FUNCTION_BLOCK FB_Tc3EventRead IMPLEMENTS InterfaceEventViewer
VAR CONSTANT
	DISP_ROWS : UDINT := 80;
END_VAR
VAR_INPUT
	tzinfo : ST_TimeZoneInformation;
END_VAR
VAR_OUTPUT
	stAlarmEvents	: ARRAY [1..DISP_ROWS] OF ST_ReadEventW;
	stAlarmhistory 	: ARRAY [1..DISP_ROWS] OF ST_ReadEventW;
END_VAR
VAR
	row : UDINT := 1;
END_VAR

METHOD PRIVATE _create_current_table : BOOL
VAR_INPUT
	event_container : REFERENCE TO EventContainer;
	row		: UDINT;
	stDate	: STRING;
	stTime	: STRING;
END_VAR
VAR_INST
	iso_datetime : STRING;
END_VAR
stAlarmEvents[row].sComputer := 'Computer';
stAlarmEvents[row].sSource := 'Source';

stAlarmEvents[row].bConfirmable := event_container.event.eConfirmationState <> TcEventConfirmationState.NotSupported;
CASE event_container.event.eSeverity OF 
	TcEventSeverity.Critical:
		stAlarmEvents[row].nClass := Tc2EventClass.TCEVENTCLASS_PARAMERROR;		
	TcEventSeverity.Error:
		stAlarmEvents[row].nClass := Tc2EventClass.TCEVENTCLASS_ALARM;
	TcEventSeverity.Info:
		stAlarmEvents[row].nClass := Tc2EventClass.TCEVENTCLASS_STATEINFO;
	TcEventSeverity.Verbose:
		stAlarmEvents[row].nClass := Tc2EventClass.TCEVENTCLASS_MESSAGE;
	TcEventSeverity.Warning:
		stAlarmEvents[row].nClass := Tc2EventClass.TCEVENTCLASS_WARNING;
END_CASE

stAlarmEvents[row].nConfirmState := event_container.event.eConfirmationState;
stAlarmEvents[row].nEventId := event_container.event.nEventId;
stAlarmEvents[row].sMessageText := event_container.event_text;


iso_datetime := FILETIME64_TO_ISO8601(
					fileTime := event_container.event.nTimeRaised,
					nBias := TO_INT(tzInfo.bias), 
					bUTC :=TRUE, 
					nPrecision := 0
				);
stAlarmEvents[row].sDate := MID(iso_datetime, 10, 1);
stAlarmEvents[row].sTime := MID(iso_datetime, 8, 12);
END_METHOD

{warning 'add method implementation '}
METHOD clear : BOOL
row := 1;
MEMSET(ADR(stAlarmEvents), 0, SIZEOF(stAlarmEvents));
END_METHOD

METHOD show : BOOL
VAR_INPUT
	event_container : REFERENCE TO EventContainer;
END_VAR
VAR_INST
	iso_datetime : STRING;
END_VAR
VAR
	stDate	: STRING;
	stTime	: STRING;
END_VAR
IF NOT __ISVALIDREF(event_container) OR row > DISP_ROWS THEN
	show := TRUE;
	RETURN;
END_IF

iso_datetime := FILETIME64_TO_ISO8601(
					fileTime := event_container.event.nTimeRaised,
					nBias := TO_INT(tzInfo.bias), 
					bUTC :=TRUE, 
					nPrecision := 0
				);

stDate := MID(iso_datetime, 10, 1);
stTime := MID(iso_datetime, 8, 12);

_create_current_table(event_container, row, stDate, stTime);
			
row := row + 1;
show := FALSE;
END_METHOD

END_FUNCTION_BLOCK

(* stored: Version 1.1.0.1, ProductVersion 3.1.4024.15
   POU FB_Tc3EventRead: Id {037aed9e-3ff5-4d2c-aad1-5efc5a7a5632}, SpecialFunc None
   Method _create_current_table: Id {68bb58e5-9921-4bf5-9711-a031fb36b796}
   Method clear: Id {67504af2-00d8-40a8-85f5-8d6225afe6eb}
   Method show: Id {0c22d4db-f791-4aef-8e7f-c26c35c4cd8d} *)
